// TIA Portal V18 export
// export: Created 2026-06-08T16:32:21.300166Z, ExportSetting WithDefaults, DisplayName Totally Integrated Automation Portal, DisplayVersion V18, DisplayName TIA Portal Openness, DisplayVersion V18, DisplayName TIA Portal Version Control Interface, DisplayVersion V18, DisplayName STEP 7 Professional, DisplayVersion V18, DisplayName STEP 7 Safety, DisplayVersion V18, DisplayName WinCC Professional, DisplayVersion V18
DATA_BLOCK "BASE_SORTING_STATION_DB"   // DB28
VERSION : 0.1
// stored: AutoNumber true, InstanceOfName BASE_SORTING_STATION, InstanceOfType FB
"BASE_SORTING_STATION"
BEGIN
END_DATA_BLOCK
